{attribute addProperty BoxType "EL2502-0010-0020"}
{attribute addProperty Id "StatusAT %I*Status_59B57038162"}
{attribute addProperty CRC "4040006875"}
{attribute addProperty SizeInBites "16"}
{attribute addProperty SizeInBytes "2"}
TYPE PWM_Inputs_Channel_F0CD9CDB :
STRUCT
	{attribute addProperty Name "Status"}
	Status AT %I* : Status_59B57038;
END_STRUCT
END_TYPE

(* stored: Version 1.2.0.0, ProductVersion 3.1.4024.9
   DUT PWM_Inputs_Channel_F0CD9CDB: Id {943dcb0e-9783-4a93-a5b6-0bb104771024} *)
